// TwinCAT 3 PLC project Practice
// ProgramVersion: 3.1.4024.0
// libraries:
//   Tc2_Standard, * (Beckhoff Automation GmbH)
//   Tc2_System, * (Beckhoff Automation GmbH)
//   Tc3_Module, * (Beckhoff Automation GmbH)
// project tree:
//   DUTs/ ST_SampleValue.TcDUT
//   / PlcTask.TcTTO
//   POUs/ FB_Motor.TcPOU, F_UpdateUsingVAR.TcPOU, F_UpdateValue.TcPOU, MAIN.TcPOU
// (motion and I/O tree: see PLC project helloworld)
// real-time tasks:
//   TASK PlcTask: cycle T#10ms, priority 20, ADS port 350
//   TASK PlcTask1: cycle T#10ms, priority 21, ADS port 352

CONFIGURATION Practice
    RESOURCE PLC ON TwinCAT3
        TASK PlcTask(INTERVAL := T#10ms, PRIORITY := 21);
        PROGRAM MAIN WITH PlcTask : MAIN;
    END_RESOURCE
END_CONFIGURATION

// ---- DUTs/ST_SampleValue.TcDUT
TYPE ST_SampleValue :
STRUCT
	nNumber : DINT;
END_STRUCT
END_TYPE

// ---- POUs/MAIN.TcPOU
PROGRAM MAIN
VAR
	stStructure : ST_SampleValue;
	bFlag : BOOL := FALSE;
	nNum : DINT := 0;
	fbMotor : FB_Motor;
END_VAR

IF NOT bFlag THEN

bFlag := TRUE;
END_IF
F_UpdateValue(stStructure);
F_UpdateUsingVAR(nNUM);

END_PROGRAM

// ---- POUs/FB_Motor.TcPOU
FUNCTION_BLOCK FB_Motor
VAR_INPUT
END_VAR
VAR_OUTPUT
END_VAR
VAR
	
END_VAR

END_FUNCTION_BLOCK

// ---- POUs/F_UpdateValue.TcPOU
FUNCTION F_UpdateValue
VAR_INPUT
	stValueStructure : REFERENCE TO ST_SampleValue;
END_VAR
VAR
END_VAR

stValueStructure.nNumber := stValueStructure.nNumber + 1;

END_FUNCTION

// ---- POUs/F_UpdateUsingVAR.TcPOU
FUNCTION F_UpdateUsingVAR : BOOL
VAR_IN_OUT
	nNumber1 : DINT;
END_VAR
VAR
END_VAR

nNumber1 := nNumber1 + 1;

END_FUNCTION
